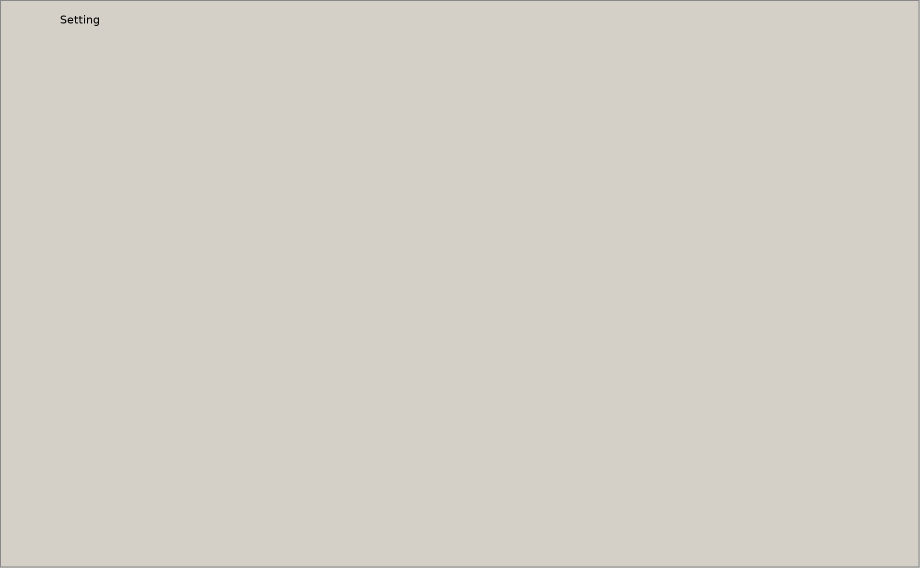
VISUALIZATION Setting  // 920x568
    Label (5,5 150x30), "Setting"
END_VISUALIZATION

(* stored: Version 1.1.0.1
   Visu Setting: Id {183cea85-788e-44d3-b990-c6aaa801135e} *)
